FUNCTION_BLOCK FB_Transport
VAR_INPUT
	bSens1 : BOOL;
	bSens2 : BOOL;
	bSens3 : BOOL;
END_VAR
VAR_OUTPUT
END_VAR
VAR
END_VAR

END_FUNCTION_BLOCK

(* stored: Version 1.1.0.1
   POU FB_Transport: Id {eef083c8-6ee7-4e91-bcb5-231fbd342ad0}, SpecialFunc None *)
